// TIA Portal V17 export
// export: Created 2025-03-05T08:02:47.0856402Z, ExportSetting WithDefaults, DisplayName Totally Integrated Automation Portal, DisplayVersion V17 Update 8, DisplayName TIA Portal Openness, DisplayVersion V17 Update 8, DisplayName TIA Portal Version Control Interface, DisplayVersion V17, DisplayName SINAMICS Startdrive Advanced, DisplayVersion V17 SP2, DisplayName SINAMICS Startdrive G110M, G120, G120C, G120D, G120P, G115D, DisplayVersion V17 SP2, DisplayName SINAMICS Startdrive G130, G150, S120, S150, SINAMICS MV, S210, DisplayVersion V17 SP2, DisplayName STEP 7 Professional, DisplayVersion V17 Update 8, DisplayName SINUMERIK ONE STEP 7 Toolbox, DisplayVersion V17 Update 12, DisplayName SINUMERIK 840D sl STEP 7 Toolbox, DisplayVersion V17 Update 12, DisplayName STEP 7 Safety, DisplayVersion V17 Update 6, DisplayName WinCC Advanced, DisplayVersion V17 Update 8
FUNCTION "FC2141_HOPPERS_LAMPS" : Void   // FC2141, LAD
{ S7_Optimized_Access := 'FALSE' }
AUTHOR : ETXETAR
VERSION : 1.0
// stored: AutoNumber false, IsIECCheckEnabled false, SetENOAutomatically false, UDAEnableTagReadback false
   VAR_TEMP
      ONE : Int;
      RETVAL1 : Int;
      SIMU_PANEL_HMI_SEL : Bool;   // SIMULATED PANEL IN HMI SELECTED
   END_VAR
   VAR CONSTANT
      FC_NUMBER : DInt := 2141;   // FC NUMBER
   END_VAR
BEGIN

REGION Network 1: LAMP - CONTROL ON
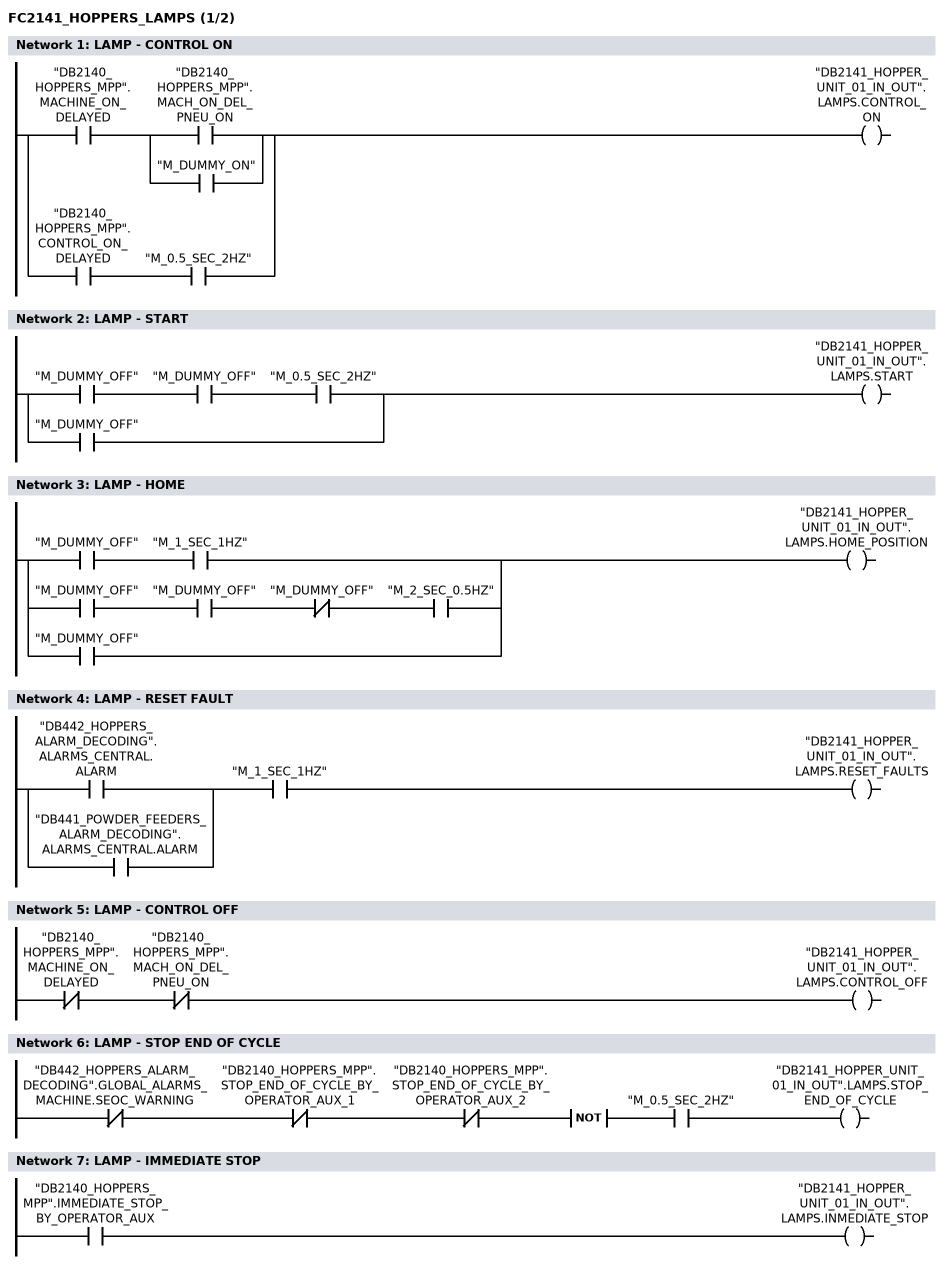
   RUNG wire#powerrail
      Contact( "DB2140_HOPPERS_MPP".MACHINE_ON_DELAYED )
      wire#w1
      Contact( "DB2140_HOPPERS_MPP".MACH_ON_DEL_PNEU_ON )
      wire#w2
      Coil( "DB2141_HOPPER_UNIT_01_IN_OUT".LAMPS.CONTROL_ON )
   END_RUNG
   RUNG wire#w1
      Contact( "M_DUMMY_ON" )
   END_RUNG wire#w2
   RUNG wire#powerrail
      Contact( "DB2140_HOPPERS_MPP".CONTROL_ON_DELAYED )
      Contact( "M_0.5_SEC_2HZ" )
   END_RUNG wire#w2
   // the same network as SCL:
   "DB2141_HOPPER_UNIT_01_IN_OUT".LAMPS.CONTROL_ON := ("DB2140_HOPPERS_MPP".MACHINE_ON_DELAYED AND ("DB2140_HOPPERS_MPP".MACH_ON_DEL_PNEU_ON OR "M_DUMMY_ON")) OR ("DB2140_HOPPERS_MPP".CONTROL_ON_DELAYED AND "M_0.5_SEC_2HZ");
END_REGION

REGION Network 2: LAMP - START
   RUNG wire#powerrail
      Contact( "M_DUMMY_OFF" )
      Contact( "M_DUMMY_OFF" )
      Contact( "M_0.5_SEC_2HZ" )
      wire#w1
      Coil( "DB2141_HOPPER_UNIT_01_IN_OUT".LAMPS.START )
   END_RUNG
   RUNG wire#powerrail
      Contact( "M_DUMMY_OFF" )
   END_RUNG wire#w1
   // the same network as SCL:
   "DB2141_HOPPER_UNIT_01_IN_OUT".LAMPS.START := ("M_DUMMY_OFF" AND "M_DUMMY_OFF" AND "M_0.5_SEC_2HZ") OR "M_DUMMY_OFF";
END_REGION

REGION Network 3: LAMP - HOME
   RUNG wire#powerrail
      Contact( "M_DUMMY_OFF" )
      Contact( "M_1_SEC_1HZ" )
      wire#w1
      Coil( "DB2141_HOPPER_UNIT_01_IN_OUT".LAMPS.HOME_POSITION )
   END_RUNG
   RUNG wire#powerrail
      Contact( "M_DUMMY_OFF" )
      Contact( "M_DUMMY_OFF" )
      I_Contact( "M_DUMMY_OFF" )
      Contact( "M_2_SEC_0.5HZ" )
   END_RUNG wire#w1
   RUNG wire#powerrail
      Contact( "M_DUMMY_OFF" )
   END_RUNG wire#w1
   // the same network as SCL:
   "DB2141_HOPPER_UNIT_01_IN_OUT".LAMPS.HOME_POSITION := ("M_DUMMY_OFF" AND "M_1_SEC_1HZ") OR ("M_DUMMY_OFF" AND "M_DUMMY_OFF" AND NOT "M_DUMMY_OFF" AND "M_2_SEC_0.5HZ") OR "M_DUMMY_OFF";
END_REGION

REGION Network 4: LAMP - RESET FAULT
   RUNG wire#powerrail
      Contact( "DB442_HOPPERS_ALARM_DECODING".ALARMS_CENTRAL.ALARM )
      wire#w1
      Contact( "M_1_SEC_1HZ" )
      Coil( "DB2141_HOPPER_UNIT_01_IN_OUT".LAMPS.RESET_FAULTS )
   END_RUNG
   RUNG wire#powerrail
      Contact( "DB441_POWDER_FEEDERS_ALARM_DECODING".ALARMS_CENTRAL.ALARM )
   END_RUNG wire#w1
   // the same network as SCL:
   "DB2141_HOPPER_UNIT_01_IN_OUT".LAMPS.RESET_FAULTS := ("DB442_HOPPERS_ALARM_DECODING".ALARMS_CENTRAL.ALARM OR "DB441_POWDER_FEEDERS_ALARM_DECODING".ALARMS_CENTRAL.ALARM) AND "M_1_SEC_1HZ";
END_REGION

REGION Network 5: LAMP - CONTROL OFF
   RUNG wire#powerrail
      I_Contact( "DB2140_HOPPERS_MPP".MACHINE_ON_DELAYED )
      I_Contact( "DB2140_HOPPERS_MPP".MACH_ON_DEL_PNEU_ON )
      Coil( "DB2141_HOPPER_UNIT_01_IN_OUT".LAMPS.CONTROL_OFF )
   END_RUNG
   // the same network as SCL:
   "DB2141_HOPPER_UNIT_01_IN_OUT".LAMPS.CONTROL_OFF := NOT "DB2140_HOPPERS_MPP".MACHINE_ON_DELAYED AND NOT "DB2140_HOPPERS_MPP".MACH_ON_DEL_PNEU_ON;
END_REGION

REGION Network 6: LAMP - STOP END OF CYCLE
   RUNG wire#powerrail
      I_Contact( "DB442_HOPPERS_ALARM_DECODING".GLOBAL_ALARMS_MACHINE.SEOC_WARNING )
      I_Contact( "DB2140_HOPPERS_MPP".STOP_END_OF_CYCLE_BY_OPERATOR_AUX_1 )
      I_Contact( "DB2140_HOPPERS_MPP".STOP_END_OF_CYCLE_BY_OPERATOR_AUX_2 )
      Not()
      Contact( "M_0.5_SEC_2HZ" )
      Coil( "DB2141_HOPPER_UNIT_01_IN_OUT".LAMPS.STOP_END_OF_CYCLE )
   END_RUNG
   // the same network as SCL:
   "DB2141_HOPPER_UNIT_01_IN_OUT".LAMPS.STOP_END_OF_CYCLE := NOT (NOT "DB442_HOPPERS_ALARM_DECODING".GLOBAL_ALARMS_MACHINE.SEOC_WARNING AND NOT "DB2140_HOPPERS_MPP".STOP_END_OF_CYCLE_BY_OPERATOR_AUX_1 AND NOT "DB2140_HOPPERS_MPP".STOP_END_OF_CYCLE_BY_OPERATOR_AUX_2) AND "M_0.5_SEC_2HZ";
END_REGION

REGION Network 7: LAMP - IMMEDIATE STOP
   RUNG wire#powerrail
      Contact( "DB2140_HOPPERS_MPP".IMMEDIATE_STOP_BY_OPERATOR_AUX )
      Coil( "DB2141_HOPPER_UNIT_01_IN_OUT".LAMPS.INMEDIATE_STOP )
   END_RUNG
   // the same network as SCL:
   "DB2141_HOPPER_UNIT_01_IN_OUT".LAMPS.INMEDIATE_STOP := "DB2140_HOPPERS_MPP".IMMEDIATE_STOP_BY_OPERATOR_AUX;
END_REGION

REGION Network 8: LAMPS - MODES
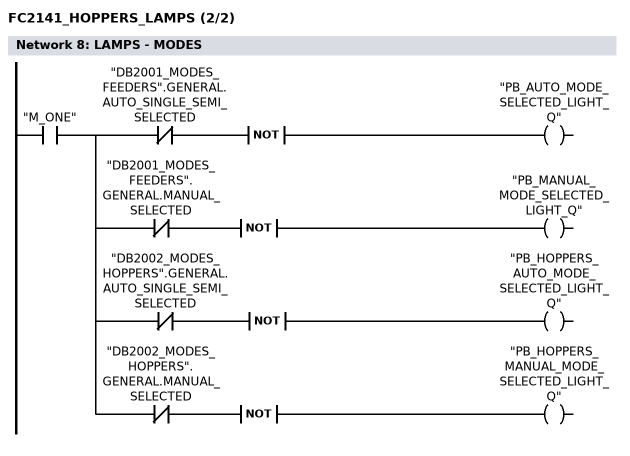
   RUNG wire#powerrail
      Contact( "M_ONE" )
      wire#w1
      I_Contact( "DB2001_MODES_FEEDERS".GENERAL.AUTO_SINGLE_SEMI_SELECTED )
      Not()
      Coil( "PB_AUTO_MODE_SELECTED_LIGHT_Q" )
   END_RUNG
   RUNG wire#w1
      I_Contact( "DB2001_MODES_FEEDERS".GENERAL.MANUAL_SELECTED )
      Not()
      Coil( "PB_MANUAL_MODE_SELECTED_LIGHT_Q" )
   END_RUNG
   RUNG wire#w1
      I_Contact( "DB2002_MODES_HOPPERS".GENERAL.AUTO_SINGLE_SEMI_SELECTED )
      Not()
      Coil( "PB_HOPPERS_AUTO_MODE_SELECTED_LIGHT_Q" )
   END_RUNG
   RUNG wire#w1
      I_Contact( "DB2002_MODES_HOPPERS".GENERAL.MANUAL_SELECTED )
      Not()
      Coil( "PB_HOPPERS_MANUAL_MODE_SELECTED_LIGHT_Q" )
   END_RUNG
   // the same network as SCL:
   "PB_AUTO_MODE_SELECTED_LIGHT_Q" := NOT ("M_ONE" AND NOT "DB2001_MODES_FEEDERS".GENERAL.AUTO_SINGLE_SEMI_SELECTED);
   "PB_MANUAL_MODE_SELECTED_LIGHT_Q" := NOT ("M_ONE" AND NOT "DB2001_MODES_FEEDERS".GENERAL.MANUAL_SELECTED);
   "PB_HOPPERS_AUTO_MODE_SELECTED_LIGHT_Q" := NOT ("M_ONE" AND NOT "DB2002_MODES_HOPPERS".GENERAL.AUTO_SINGLE_SEMI_SELECTED);
   "PB_HOPPERS_MANUAL_MODE_SELECTED_LIGHT_Q" := NOT ("M_ONE" AND NOT "DB2002_MODES_HOPPERS".GENERAL.MANUAL_SELECTED);
END_REGION
END_FUNCTION
